// TIA Portal V16 export
// export: Created 2024-09-05T17:40:13.6176037Z, ExportSetting WithDefaults, DisplayName Totally Integrated Automation Portal, DisplayVersion V16 Update 6, DisplayName TIA Portal Version Control Interface, DisplayVersion V16 Update 2, DisplayName TIA Portal Openness, DisplayVersion V16 Update 6, DisplayName STEP 7 Professional, DisplayVersion V16 Update 6, DisplayName STEP 7 Safety, DisplayVersion V16, DisplayName WinCC Advanced, DisplayVersion V16 Update 6
TYPE "UDT_DateTimeAndShiftsSettings"
// stored: IsFailsafeCompliant false
   STRUCT
      DateAndTime : DTL := DTL#2019-01-17-00:00:00;   // Date and time to set
      Shift1Enabled : Bool := TRUE;   // Shift 1 enabled: 0= No,
      Shift1StartTime : Time_Of_Day := TOD#6:0:0.000;   // Shift 1 start time
      Shift1EndTime : Time_Of_Day := TOD#14:0:0.000;   // Shift 1 end time
      Shift2Enabled : Bool := TRUE;   // Shift 2 enabled: 0= No
      Shift2StartTime : Time_Of_Day := TOD#14:0:0.000;   // Shift 2 start time
      Shift2EndTime : Time_Of_Day := TOD#22:0:0.000;   // Shift 2 end time
      Shift3Enabled : Bool := TRUE;   // Shift 3 enabled: 0= No
      Shift3StartTime : Time_Of_Day := TOD#22:0:0.000;   // Shift 3 start time
      Shift3EndTime : Time_Of_Day := TOD#6:0:0.000;   // Shift 3 end time
   END_STRUCT;
END_TYPE
